FUNCTION_BLOCK FB_NciChannel EXTENDS FB_ComponentBase IMPLEMENTS I_NciChannel_GCode

VAR_INPUT
    stAxisIds : ST_NciAxisIds;
	nGroupId  : UDINT := 4;
END_VAR

VAR
    // Zmienne zlinkowane bezpośrednio z hardwarem kanału NCI
    stNciToPlc AT %I* : NCTOPLC_NCICHANNEL_REF; 
    stPlcToNci AT %Q* : PLCTONC_NCICHANNEL_REF;

    // Bloki systemowe Beckhoffa do obsługi grupy
	fbBuildExtGroup : CfgBuildExt3DGroup;
    fbUngroup       : CfgReconfigGroup;
    
    // Bloki systemowe do obsługi programu i ruchu (nowe wersje Ex)
    fbLoadProg      : ItpLoadProgEx;
    fbStartStop     : ItpStartStopEx;
    fbReset         : ItpResetEx2;
    
    _IsGrouped      : BOOL;
    _IsProgLoaded   : BOOL;
    _IsReady		:BOOL;
	


END_VAR

METHOD BuildGroup
_IsGrouped := FALSE;
_Error := FALSE; 
_ErrorId := 0;

fbBuildExtGroup(
    bExecute := TRUE,
    nGroupId := nGroupId,
    nXAxisId := stAxisIds.nX,
    nYAxisId := stAxisIds.nY,
    nZAxisId := stAxisIds.nZ,
    nQ1AxisId := stAxisIds.nQ1
);
END_METHOD

PROPERTY ChannelError : BOOL
GET
ChannelError := _Error OR (stNciToPlc.ErrorCode <> 0);
END_GET
END_PROPERTY

PROPERTY ChannelErrorId : UDINT
GET
IF stNciToPlc.ErrorCode <> 0 THEN
    ChannelErrorId := stNciToPlc.ErrorCode;
ELSE
    ChannelErrorId := _ErrorId;
END_IF
END_GET
END_PROPERTY

// This method serves as the entry point for all underlying FB logic
METHOD PUBLIC CyclicLogic

// This method should be called cyclically by descendant function blocks by invoking SUPER^.CyclicLogic().  Alternatively, the contents of this method could be reimplemented entirely in which case a call to this method would not be necessary.
// Wywołanie bazowe
SUPER^.CyclicLogic();

// Odblokowanie posuwu kanału NCI (1000000 = 100%)
stPlcToNci.ChnAxesOvr := 1000000;

// --- ODŚWIEŻANIE BLOKÓW SYSTEMOWYCH ---
fbBuildExtGroup(tTimeOut := T#2S);
fbUngroup(tTimeOut := T#2S);


fbLoadProg(
    sNciToPlc := stNciToPlc, 
    tTimeOut := T#2S
);

fbStartStop(
    sNciToPlc := stNciToPlc, 
    tTimeOut := T#2S
);

fbReset(
    sNciToPlc := stNciToPlc, 
    tTimeOut := T#2S
);

// --- AKTUALIZACJA STATUSÓW ---
// Obsługa stanów dla tworzenia grupy
IF fbStartStop.bErr THEN
    _Error := TRUE;
    _ErrorId := fbStartStop.nErrId;
    fbStartStop(bStart := FALSE, bStop := FALSE, sNciToPlc := stNciToPlc);
ELSIF fbStartStop.bBusy THEN
    // Skoro kanał NCI przyjął komendę i jest zajęty, opuszczamy Start, 
    // aby przygotować blok na kolejne uruchomienie w przyszłości
    fbStartStop(bStart := FALSE, sNciToPlc := stNciToPlc);
ELSIF NOT fbStartStop.bBusy AND fbStartStop.bStop THEN
    // Jak się poprawnie zatrzymał, opuszczamy flagę Stop
    fbStartStop(bStop := FALSE, sNciToPlc := stNciToPlc);
END_IF

// Obsługa stanów dla rozpinania grupy
IF fbUngroup.bErr THEN
    _Error := TRUE;
    _ErrorId := fbUngroup.nErrId;
    fbUngroup(bExecute := FALSE);
    _IsGrouped := FALSE; // W razie błędu awaryjnie zdejmujemy flagę, żeby maszyna nie utknęła na zawsze
ELSIF fbUngroup.bBusy = FALSE AND fbUngroup.bExecute THEN
    _IsGrouped := FALSE; // Pomyślnie rozpięto!
    fbUngroup(bExecute := FALSE);
END_IF


IF fbBuildExtGroup.bErr THEN
    _Error := TRUE;
    _ErrorId := fbBuildExtGroup.nErrId;
ELSIF fbBuildExtGroup.bBusy = FALSE AND fbBuildExtGroup.bExecute THEN
    _IsGrouped := TRUE;
    fbBuildExtGroup(bExecute := FALSE);
END_IF

// Podobnie dla ładowania programu
IF fbLoadProg.bErr THEN
    _Error := TRUE;
    _ErrorId := fbLoadProg.nErrId;
ELSIF fbLoadProg.bBusy = FALSE AND fbLoadProg.bExecute THEN
    _IsProgLoaded := TRUE;
	fbLoadProg(bExecute := FALSE, sNciToPlc := stNciToPlc);
END_IF

// --- OBSŁUGA ZEROWANIA fbReset ---
IF fbReset.bErr THEN
    _Error := TRUE;
    _ErrorId := fbReset.nErrId;
    fbReset(bExecute := FALSE, sNciToPlc := stNciToPlc);
ELSIF fbReset.bBusy = FALSE AND fbReset.bExecute THEN
    fbReset(bExecute := FALSE, sNciToPlc := stNciToPlc);
END_IF
END_METHOD

PROPERTY IsGrouped : BOOL
GET
IsGrouped := _IsGrouped;
END_GET
END_PROPERTY

PROPERTY IsMoving : BOOL
GET
IsMoving := (stNciToPlc.ItpState = 5);
END_GET
END_PROPERTY

PROPERTY IsProgramLoaded : BOOL
GET
IsProgramLoaded := _IsProgLoaded;
END_GET
END_PROPERTY

PROPERTY IsReady : BOOL
GET
IsReady := (stNciToPlc.ItpState = 2);
END_GET
END_PROPERTY

METHOD LoadProgram
VAR_INPUT
	sProgramPath : STRING(255);
END_VAR
_IsProgLoaded := FALSE;
fbLoadProg(
    bExecute := TRUE,
    sPrg := sProgramPath,
    nLength := INT_TO_UDINT(LEN(sProgramPath)),
    sNciToPlc := stNciToPlc 
);
END_METHOD

METHOD ResetChannel
VAR_INPUT
END_VAR
// Najpierw bezwarunkowo ubijamy flagi ruchu
fbStartStop(bStart := FALSE, bStop := FALSE, sNciToPlc := stNciToPlc);

// Następnie resetujemy sam kanał NCI
fbReset(
    bExecute := TRUE,
    sNciToPlc := stNciToPlc
);

_Error := FALSE;
_ErrorId := 0;
END_METHOD

METHOD Start
VAR_INPUT
END_VAR
fbStartStop(
    bStart := TRUE, 
    bStop := FALSE,
    sNciToPlc := stNciToPlc 
);
END_METHOD

METHOD Stop
VAR_INPUT
END_VAR
fbStartStop(
    bStart := FALSE, 
    bStop := TRUE,
    sNciToPlc := stNciToPlc
);
END_METHOD

METHOD Ungroup
VAR_INPUT
END_VAR
fbUngroup(
    bExecute := TRUE, 
    nGroupId := nGroupId
);
END_METHOD

END_FUNCTION_BLOCK

(* stored: Version 1.1.0.1, ProductVersion 3.1.4024.15
   POU FB_NciChannel: Id {08e0b468-709d-436d-9099-2993cda1a53a}, SpecialFunc None
   Method BuildGroup: Id {66cae995-577f-4fd0-87b2-2377298b6c08}
   Property ChannelError: Id {00e4bd1a-bf02-4d2b-946a-25a3bc45656f}
   Get Get: Id {f4ebe933-f7f9-435a-92ab-18b62f7e1f3b}
   Property ChannelErrorId: Id {5eecb53c-95cd-4946-aa97-89be021e8fb6}
   Get Get: Id {b56a0d9f-fbbe-4639-aa87-9f6a3e9935e4}
   Method CyclicLogic: Id {06e1abcc-1131-428d-af2d-924cc3aee150}
   Property IsGrouped: Id {f6f0eca0-33a2-495f-820d-274c738b997a}
   Get Get: Id {d1c66ce7-95a8-4d4e-be30-7abf09c06e2e}
   Property IsMoving: Id {d2e008d1-a7d6-4d22-954d-244be66e8771}
   Get Get: Id {3e2ebb55-5f4f-4667-bd58-50412615786d}
   Property IsProgramLoaded: Id {0b92f6bd-d666-452f-8e89-937b5dadb29a}
   Get Get: Id {d292bbc4-723c-4a6a-9853-4c75c2dbf160}
   Property IsReady: Id {cf337947-e57f-47e4-be99-6e54e3f523cc}
   Get Get: Id {23882524-4a9e-4cc6-9ca4-0c5f8369503c}
   Method LoadProgram: Id {8e5b758c-dd77-4196-8305-9ba935eedf73}
   Method ResetChannel: Id {a5c8a5c9-f0bb-40f8-b374-213a9332f10f}
   Method Start: Id {4f54c653-5d61-4053-b4b3-0f559e72e12d}
   Method Stop: Id {e02489bc-47d1-4068-b1f1-be7069b73cea}
   Method Ungroup: Id {c18a5735-a574-4548-beb3-a5ca7ced70aa} *)
